FUNCTION_BLOCK FB_LUTDevice_1 EXTENDS FD_Device IMPLEMENTS ITF_Convoyer
VAR_INPUT
END_VAR

VAR_OUTPUT
END_VAR

VAR
	//=====================
	fbPneuCyl_AxisZ										: FB_PneuCyl_3Pos(
		
																										 ); 
END_VAR

VAR CONSTANT
	// --------------------------Base------------------
	C_SeqStep_OnBasePos_Start								: UINT :=  20; 
	C_SeqStep_OnBasePos_WaitOpMode					: UINT :=  30;
	C_SeqStep_OnBasePos_Done								: UINT :=  100; 
	
	// --------------------------Auto Sequence------------------
	
	C_SeqStep_Auto_Start										: UINT :=  200;
	C_SeqStep_Auto_End											: UINT :=  400;
END_VAR


//******* Important and necessary
SUPER^();  

//====================================
IF NOT Enable THEN RETURN; END_IF

//FB_Init ist immer implizit verfügbar und wird primär für die Initialisierung verwendet.
//Der Rückgabewert wird nicht ausgewertet. Für gezielte Einflussnahme können Sie
//die Methoden explizit deklarieren und darin mit dem Standard-Initialisierungscode 
//zusätzlichen Code bereitstellen. Sie können den Rückgabewert auswerten.
METHOD FB_Init: BOOL
VAR_INPUT    
	bInitRetains					: BOOL; 					// TRUE: Die Retain-Variablen werden initialisiert (Reset warm / Reset kalt)    
	bInCopyCode						: BOOL;  					// TRUE: Die Instanz wird danach in den Kopiercode kopiert (Online-Change)
	
	I_Name                : STRING;         //  Name
	I_ID                  : UINT;           // ID
  I_itfOwner					  : ITF_Owner;      // owner 
END_VAR
END_METHOD

METHOD mAutomatic : E_CmdState
VAR_INPUT
	I_bExecute	: BOOL;
END_VAR
END_METHOD

METHOD mCmdExec_Auto : UINT
VAR_INPUT
END_VAR

CASE SequenceID OF

  //******************************************************* Idle 
  C_SeqStep_Idle: 
  	SequenceID       :=  C_SeqStep_Start;
  
  //****************************************************** Start
  C_SeqStep_Start:
  	
  	SequenceID       :=  C_SeqStep_OnBasePos_Start;
	C_SeqStep_OnBasePos_Start:
	
		SequenceID       :=  C_SeqStep_Done;;
	
	C_SeqStep_OnBasePos_Start:
	;
	
	C_SeqStep_OnBasePos_Start:
	;
	
  C_SeqStep_Error: 
    //************* all FB reset

		//************* 
    mSequence := mDone(); 
  //**********************Done 
  	
 	C_SeqStep_Done:
  	mSequence := mDone();

END_CASE
END_METHOD

METHOD mCmdExec_Homing : UINT
VAR_INPUT
END_VAR

CASE SequenceID OF

  //******************************************************* Idle 
  C_SeqStep_Idle: 
  	SequenceID       :=  C_SeqStep_Start;
  
  //****************************************************** Start
  C_SeqStep_Start:
   
  	SequenceID       :=  C_SeqStep_Done;
	
  C_SeqStep_Error: 
    //************* all FB reset

		//************* 
    mSequence := mDone(); 
  //**********************Done 
  	
 	C_SeqStep_Done:
  	mSequence := mDone();

END_CASE
END_METHOD

METHOD mCmdExec_Service : UINT
VAR_INPUT
END_VAR
END_METHOD

METHOD mHold : E_CmdState
VAR_INPUT
	I_bExecute	: BOOL;
END_VAR
END_METHOD

METHOD mHome : E_CmdState
VAR_INPUT
	I_bExecute	: BOOL;
END_VAR
END_METHOD

METHOD mRelease : E_CmdState
VAR_INPUT
	I_bExecute	: BOOL;
END_VAR
END_METHOD

METHOD mSequence : E_CmdState
VAR_INPUT
	I_bExecute				: BOOL;
END_VAR

VAR
	L_eState 					: E_CmdState;
END_VAR
mSequence := SUPER^.mSequence(I_bExecute);	


// Generic checks from parent
L_eState := SUPER^.mSequence(I_bExecute := I_bExecute);

IF L_eState <> E_CmdState.Busy 
	THEN
    mSequence := L_eState;
    RETURN;
END_IF

CASE Mode OF
	E_Mode.Homing:
		mCmdExec_Homing();
		
	E_Mode.Auto:
		mCmdExec_Auto();
		
	E_Mode.Homing:
		mCmdExec_Service();
		
END_CASE
END_METHOD

METHOD mService : E_CmdState
VAR_INPUT
	I_bExecute	: BOOL;
END_VAR
END_METHOD

METHOD mStop : E_CmdState
VAR_INPUT
	I_bExecute	: BOOL;
END_VAR
END_METHOD

END_FUNCTION_BLOCK

(* stored: Version 1.1.0.1, ProductVersion 3.1.4026.18
   POU FB_LUTDevice_1: Id {5feb55c0-427c-48c9-ba35-af743a91e620}, SpecialFunc None
   Folder 01 Properties: Id {2aabb068-656d-41fd-a806-cf76b4cb3441}
   Folder 02 Methodes: Id {1506cc05-5219-4049-9dc0-2e7a95a3ee83}
   Folder 100 CmdExecute: Id {7e328eca-1401-459e-a275-f97eb30a6441}
   Method FB_Init: Id {1f043a9f-9106-4491-8db0-3f1836aec147}
   Method mAutomatic: Id {1835ff83-941d-4063-a840-8408932dddd1}
   Method mCmdExec_Auto: Id {5701aa1e-f0ac-48f8-996d-a5d08e5d82fc}
   Method mCmdExec_Homing: Id {d08c680c-f637-4787-ade1-99e01f84de11}
   Method mCmdExec_Service: Id {d21b21ff-2e17-466c-8843-dbd9bfd40883}
   Method mHold: Id {137e727c-298e-40d1-b133-78a53a4da30c}
   Method mHome: Id {241edc62-8f63-4ac6-a585-5a616b65502a}
   Method mRelease: Id {1c0b6c40-6835-4a42-92c2-94882e6246d3}
   Method mSequence: Id {6b2421d1-3f7c-46f5-b14b-e3bd2e81423d}
   Method mService: Id {769cc3db-2bac-4bc7-9880-022e0482c827}
   Method mStop: Id {edaab38f-4b09-41f6-8b05-2696db87e6da} *)
